# EPICS IOC start-up script: iocsh/sce.iocsh
# .init.iocsh
# ===========

dbLoadRecords "engine.db"       "P=$(P)"
dbLoadRecords "gplug.db"        "P=$(P), PG=$(PG)"
dbLoadRecords "io.db"           "P=$(P)"
dbLoadRecords "iosingle.db"     "P=$(P)"
dbLoadRecords "ctrl.db"         "P=$(P)"
dbLoadRecords "states.db"       "P=$(P)"

mapStrOut "databufferLink"      "$(DBUFL)"
mapStrOut "mevtsLink"           "$(MEVTSL)"
mapStrOut "sctableRoot"         "$(SCTROOT)"

var "iodebug" "4"
#var PscUs 888

#EOF
